(* Logix 5000 project; controller Comas_L4 vendor 1 type 14 code 193 rev 30.11; software revision 30.02; part 3 of 12 *)

ADD_ON_INSTRUCTION Message_Axe   (* revision 1.1 *)
VAR_IN_OUT
   MIO_Axis : AXIS_CIP_DRIVE; {required}
   Inf_Messages : STRING[380]; {required}
END_VAR
VAR_OUTPUT
   ER : BOOL; {access Read Only, visible}
END_VAR
VAR_IN_OUT
   Message_Defaut : STRING; {required}
   L_Msg_Index : DINT; {required}
END_VAR
VAR
   TRUE : BOOL := 1;
   FALSE : BOOL;
   L_MemoResultIndex : DINT; {access None}
   Numero_Texte : DINT; {access Read Only}
END_VAR

ROUTINE Logic   (* structured text *)
   
   	(*----------------------------------------------------------------------------------------------------
   										Build Axis ResultText String Info
   	-----------------------------------------------------------------------------------------------------*)
   		IF L_MemoResultIndex <> L_Msg_Index THEN
   			COP(Inf_Messages[L_Msg_Index],Message_Defaut,1);
   			L_MemoResultIndex					:= L_Msg_Index;
   		END_IF;
   (*================================================================================================
   										CHECK FAULT
   ==================================================================================================*)
   IF MIO_Axis.AxisFault <> 0 THEN
   
   	(*================================================================================================
   									Physical Axis Fault
   	==================================================================================================*)
   	IF MIO_Axis.AxisFault.0 THEN
   		(*================================================================================================
   										MOTOR COMMUTATION FAULT
   			==================================================================================================*)
   			IF 		MIO_Axis.MotorCommutationFault THEN
   			 		L_Msg_Index													:= 134;							// Convert INT_To_DINT
   					Numero_Texte														:= 2000+ L_Msg_Index;			// Class 2 Fault
   			(*================================================================================================
   										MOTOR OVERSEPEED FL FAULT
   			==================================================================================================*)
   			ELSIF 	MIO_Axis.MotorOverspeedFLFault THEN
   			 		L_Msg_Index													:= 135;							// Convert INT_To_DINT
   					Numero_Texte														:= 2000+ L_Msg_Index;			// Class 2 Faultt
   			(*================================================================================================
   										MOTOR OVERSEPEED UL FAULT
   			==================================================================================================*)
   			ELSIF 	MIO_Axis.MotorOverspeedULFault THEN
   			 		L_Msg_Index													:= 136;							// Convert INT_To_DINT
   					Numero_Texte														:= 2000+ L_Msg_Index;			// Class 2 Faultt
   			(*================================================================================================
   										MOTOR OVERTEMPERATURE FL FAULT
   			==================================================================================================*)
   			ELSIF 	MIO_Axis.MotorOvertemperatureFLFault THEN
   			 		L_Msg_Index													:= 137;							// Convert INT_To_DINT
   					Numero_Texte														:= 2000+ L_Msg_Index;			// Class 2 Faultt
   			(*================================================================================================
   										MOTOR OVERTEMPERATURE UL FAULT
   			==================================================================================================*)
   			ELSIF 	MIO_Axis.MotorOvertemperatureULFault THEN
   			 		L_Msg_Index													:= 138;							// Convert INT_To_DINT
   					Numero_Texte														:= 2000+ L_Msg_Index;			// Class 2 Faultt
   			(*================================================================================================
   										MOTOR THERMAL OVERLOAD FL FAULT
   			==================================================================================================*)
   			ELSIF 	MIO_Axis.MotorThermalOverloadFLFault THEN
   			 		L_Msg_Index													:= 139;							// Convert INT_To_DINT
   					Numero_Texte														:= 2000+ L_Msg_Index;			// Class 2 Faultt
   			(*================================================================================================
   										MOTOR THERMAL OVERLOAD UL FAULT
   			==================================================================================================*)
   			ELSIF 	MIO_Axis.MotorThermalOverloadULFault THEN
   			 		L_Msg_Index													:= 140;							// Convert INT_To_DINT
   					Numero_Texte														:= 2000+ L_Msg_Index;			// Class 2 Faultt
   			(*================================================================================================
   										INVERTER OVERCURRENT FAULT
   			==================================================================================================*)
   			ELSIF 	MIO_Axis.InverterOvercurrentFault THEN
   			 		L_Msg_Index													:= 141;							// Convert INT_To_DINT
   					Numero_Texte														:= 2000+ L_Msg_Index;			// Class 2 Faultt
   			(*================================================================================================
   										INVERTER OVERTEMPERATURE FL FAULT
   			==================================================================================================*)
   			ELSIF 	MIO_Axis.InverterOvertemperatureFLFault THEN
   			 		L_Msg_Index													:= 142;							// Convert INT_To_DINT
   					Numero_Texte														:= 2000+ L_Msg_Index;			// Class 2 Faultt
   			(*================================================================================================
   										INVERTER OVERTEMPERATURE UL FAULT
   			==================================================================================================*)
   			ELSIF 	MIO_Axis.InverterOvertemperatureULFault THEN
   			 		L_Msg_Index													:= 143;							// Convert INT_To_DINT
   					Numero_Texte														:= 2000+ L_Msg_Index;			// Class 2 Faultt
   			(*================================================================================================
   										INVERTER THERMALOVERLOAD FL FAULT
   			==================================================================================================*)
   			ELSIF 	MIO_Axis.InverterThermalOverloadFLFault THEN
   			 		L_Msg_Index													:= 144;							// Convert INT_To_DINT
   					Numero_Texte														:= 2000+ L_Msg_Index;			// Class 2 Faultt
   			(*================================================================================================
   										INVERTER OVERTEMPERATURE UL FAULT
   			==================================================================================================*)
   			ELSIF 	MIO_Axis.InverterOvertemperatureULFault THEN
   			 		L_Msg_Index													:= 145;							// Convert INT_To_DINT
   					Numero_Texte														:= 2000+ L_Msg_Index;			// Class 2 Faultt
   			(*================================================================================================
   										CONVERTER GROUND CURRENT FL FAULT
   			==================================================================================================*)
   			ELSIF 	MIO_Axis.ConverterGroundCurrentFLFault THEN
   			 		L_Msg_Index													:= 146;							// Convert INT_To_DINT
   					Numero_Texte														:= 2000+ L_Msg_Index;			// Class 2 Faultt
   			(*================================================================================================
   										CONVERTER GROUND CURRENT UL FAULT
   			==================================================================================================*)
   			ELSIF 	MIO_Axis.ConverterGroundCurrentULFault THEN
   			 		L_Msg_Index													:= 147;							// Convert INT_To_DINT
   					Numero_Texte														:= 2000+ L_Msg_Index;			// Class 2 Faultt
   			(*================================================================================================
   										CONVERTER OVERTEMPERATURE FL FAULT
   			==================================================================================================*)
   			ELSIF 	MIO_Axis.ConverterOvertemperatureFLFault THEN
   			 		L_Msg_Index													:= 148;							// Convert INT_To_DINT
   					Numero_Texte														:= 2000+ L_Msg_Index;			// Class 2 Faultt
   			(*================================================================================================
   										CONVERTER OVERTEMPERATURE UL FAULT
   			==================================================================================================*)
   			ELSIF 	MIO_Axis.ConverterOvertemperatureULFault THEN
   			 		L_Msg_Index													:= 149;							// Convert INT_To_DINT
   					Numero_Texte														:= 2000+ L_Msg_Index;			// Class 2 Faultt
   			(*================================================================================================
   										CONVERTER THERMAL OVERLOAD FL FAULT
   			==================================================================================================*)
   			ELSIF 	MIO_Axis.ConverterThermalOverloadFLFault THEN
   			 		L_Msg_Index													:= 150;							// Convert INT_To_DINT
   					Numero_Texte														:= 2000+ L_Msg_Index;			// Class 2 Faultt
   			(*================================================================================================
   										CONVERTER THERMAL OVERLOAD UL FAULT
   			==================================================================================================*)
   			ELSIF 	MIO_Axis.ConverterThermalOverloadULFault THEN
   			 		L_Msg_Index													:= 151;							// Convert INT_To_DINT
   					Numero_Texte														:= 2000+ L_Msg_Index;			// Class 2 Faultt
   			(*================================================================================================
   										CONVERTER AC POWER LOSS FAULT
   			==================================================================================================*)
   			ELSIF 	MIO_Axis.ConverterACPowerLossFault THEN
   			 		L_Msg_Index													:= 152;							// Convert INT_To_DINT
   					Numero_Texte														:= 2000+ L_Msg_Index;			// Class 2 Faultt
   			(*================================================================================================
   										CONVERTER AC SINGLE PHASE LOSS FAULT
   			==================================================================================================*)
   			ELSIF 	MIO_Axis.ConverterACSinglePhaseLossFault THEN
   			 		L_Msg_Index													:= 153;							// Convert INT_To_DINT
   					Numero_Texte														:= 2000+ L_Msg_Index;			// Class 2 Faultt
   			(*================================================================================================
   										CONVERTER AC PHASE SHORT FAULT
   			==================================================================================================*)
   			ELSIF 	MIO_Axis.ConverterACPhaseShortFault THEN
   			 		L_Msg_Index													:= 154;							// Convert INT_To_DINT
   					Numero_Texte														:= 2000+ L_Msg_Index;			// Class 2 Faultt
   			(*================================================================================================
   										CONVERTER PRE CHARGE FAULT
   			==================================================================================================*)
   			ELSIF 	MIO_Axis.ConverterACSinglePhaseLossFault THEN
   			 		L_Msg_Index													:= 155;							// Convert INT_To_DINT
   					Numero_Texte														:= 2000+ L_Msg_Index;			// Class 2 Faultt
   			(*================================================================================================
   										BUS REGULATOR OVERTEMPERATURE FL FAULT
   			==================================================================================================*)
   			ELSIF 	MIO_Axis.BusRegulatorOvertemperatureFLFault THEN
   			 		L_Msg_Index													:= 156;							// Convert INT_To_DINT
   					Numero_Texte														:= 2000+ L_Msg_Index;			// Class 2 Faultt
   			(*================================================================================================
   										BUS REGULATOR OVERTEMPERATURE UL FAULT
   			==================================================================================================*)
   			ELSIF 	MIO_Axis.BusRegulatorOvertemperatureULFault THEN
   			 		L_Msg_Index													:= 157;							// Convert INT_To_DINT
   					Numero_Texte														:= 2000+ L_Msg_Index;			// Class 2 Faultt
   			(*================================================================================================
   										BUS REGULATOR THERMAL OVERLOAD FL FAULT
   			==================================================================================================*)
   			ELSIF 	MIO_Axis.BusRegulatorThermalOverloadFLFault THEN
   			 		L_Msg_Index													:= 158;							// Convert INT_To_DINT
   					Numero_Texte														:= 2000+ L_Msg_Index;			// Class 2 Faultt
   			(*================================================================================================
   										BUS REGULATOR THERMAL OVERLOAD UL FAULT
   			==================================================================================================*)
   			ELSIF 	MIO_Axis.BusRegulatorThermalOverloadULFault THEN
   			 		L_Msg_Index													:= 159;							// Convert INT_To_DINT
   					Numero_Texte														:= 2000+ L_Msg_Index;			// Class 2 Faultt
   			(*================================================================================================
   										BUS UNDERVOLTAGE FL FAULT
   			==================================================================================================*)
   			ELSIF 	MIO_Axis.BusUndervoltageFLFault THEN
   			 		L_Msg_Index													:= 160;							// Convert INT_To_DINT
   					Numero_Texte														:= 2000+ L_Msg_Index;			// Class 2 Faultt
   			(*================================================================================================
   										BUS UNDERVOLTAGE UL FAULT
   			==================================================================================================*)
   			ELSIF 	MIO_Axis.BusUndervoltageULFault THEN
   			 		L_Msg_Index													:= 161;							// Convert INT_To_DINT
   					Numero_Texte														:= 2000+ L_Msg_Index;			// Class 2 Faultt
   			(*================================================================================================
   										BUS OVERVOLTAGE FL FAULT
   			==================================================================================================*)
   			ELSIF 	MIO_Axis.BusOvervoltageFLFault THEN
   			 		L_Msg_Index													:= 162;							// Convert INT_To_DINT
   					Numero_Texte														:= 2000+ L_Msg_Index;			// Class 2 Faultt
   			(*================================================================================================
   										BUS OVERVOLTAGE UL FAULT
   			==================================================================================================*)
   			ELSIF 	MIO_Axis.BusOvervoltageULFault THEN
   			 		L_Msg_Index													:= 163;							// Convert INT_To_DINT
   					Numero_Texte														:= 2000+ L_Msg_Index;			// Class 2 Faultt
   			(*================================================================================================
   										BUS POWER LOSS FAULT
   			==================================================================================================*)
   			ELSIF 	MIO_Axis.BusPowerLossFault THEN
   			 		L_Msg_Index													:= 164;							// Convert INT_To_DINT
   					Numero_Texte														:= 2000+ L_Msg_Index;			// Class 2 Faultt
   			(*================================================================================================
   										BUS POWER BLOWN FUSE FAULT
   			==================================================================================================*)
   			ELSIF 	MIO_Axis.BusPowerBlownFuseFault THEN
   			 		L_Msg_Index													:= 165;							// Convert INT_To_DINT
   					Numero_Texte														:= 2000+ L_Msg_Index;			// Class 2 Faultt
   			(*================================================================================================
   										FEEDBACK SIGNAL NOISE FL FAULT
   			==================================================================================================*)
   			ELSIF 	MIO_Axis.FeedbackSignalNoiseFLFault THEN
   			 		L_Msg_Index													:= 166;							// Convert INT_To_DINT
   					Numero_Texte														:= 2000+ L_Msg_Index;			// Class 2 Faultt
   			(*================================================================================================
   										FEEDBACK SIGNAL NOISE UL FAULT
   			==================================================================================================*)
   			ELSIF 	MIO_Axis.FeedbackSignalNoiseULFault THEN
   			 		L_Msg_Index													:= 167;							// Convert INT_To_DINT
   					Numero_Texte														:= 2000+ L_Msg_Index;			// Class 2 Faultt
   			(*================================================================================================
   										FEEDBACK SIGNAL LOSS FL FAULT
   			==================================================================================================*)
   			ELSIF 	MIO_Axis.FeedbackSignalLossFLFault THEN
   			 		L_Msg_Index													:= 168;							// Convert INT_To_DINT
   					Numero_Texte														:= 2000+ L_Msg_Index;			// Class 2 Faultt
   			(*================================================================================================
   										FEEDBACK SIGNAL LOSS UL FAULT
   			==================================================================================================*)
   			ELSIF 	MIO_Axis.FeedbackSignalLossULFault THEN
   			 		L_Msg_Index													:= 169;							// Convert INT_To_DINT
   					Numero_Texte														:= 2000+ L_Msg_Index;			// Class 2 Faultt
   			(*================================================================================================
   										FEEDBACK DATA LOSS FL FAULT
   			==================================================================================================*)
   			ELSIF 	MIO_Axis.FeedbackDataLossFLFault THEN
   			 		L_Msg_Index													:= 170;							// Convert INT_To_DINT
   					Numero_Texte														:= 2000+ L_Msg_Index;			// Class 2 Faultt
   			(*================================================================================================
   										FEEDBACK DATA LOSS UL FAULT
   			==================================================================================================*)
   			ELSIF 	MIO_Axis.FeedbackDataLossULFault THEN
   			 		L_Msg_Index													:= 171;							// Convert INT_To_DINT
   					Numero_Texte														:= 2000+ L_Msg_Index;			// Class 2 Faultt
   			(*================================================================================================
   										FEEDBACK DEVICE FAULT
   			==================================================================================================*)
   			ELSIF 	MIO_Axis.FeedbackDeviceFault THEN
   			 		L_Msg_Index													:= 172;							// Convert INT_To_DINT
   					Numero_Texte														:= 2000+ L_Msg_Index;			// Class 2 Faultt
   			(*================================================================================================
   										HARDWARE OVERTRAVEL POSITIVE FAULT
   			==================================================================================================*)
   			ELSIF 	MIO_Axis.HardwareOvertravelPositiveFault THEN
   			 		L_Msg_Index													:= 173;							// Convert INT_To_DINT
   					Numero_Texte														:= 2000+ L_Msg_Index;			// Class 2 Faultt
   			(*================================================================================================
   										HARDWARE OVERTRAVEL NEGATIVE FAULT
   			==================================================================================================*)
   			ELSIF 	MIO_Axis.HardwareOvertravelNegativeFault THEN
   			 		L_Msg_Index													:= 174;							// Convert INT_To_DINT
   					Numero_Texte														:= 2000+ L_Msg_Index;			// Class 2 Faultt
   			(*================================================================================================
   										EXCESSIVE POSITION ERROR FAULT
   			==================================================================================================*)
   			ELSIF 	MIO_Axis.ExcessivePositionErrorFault	THEN
   			 		L_Msg_Index													:= 175;							// Convert INT_To_DINT
   					Numero_Texte														:= 2000+ L_Msg_Index;			// Class 2 Faultt
   			(*================================================================================================
   										EXCESSIVE VELOCITY ERROR FAULT
   			==================================================================================================*)
   			ELSIF 	MIO_Axis.ExcessiveVelocityErrorFault	THEN
   			 		L_Msg_Index													:= 176;							// Convert INT_To_DINT
   					Numero_Texte														:= 2000+ L_Msg_Index;			// Class 2 Faultt
   			(*================================================================================================
   										OVERTORQUE LIMIT FAULT
   			==================================================================================================*)
   			ELSIF 	MIO_Axis.OvertorqueLimitFault	THEN
   			 		L_Msg_Index													:= 177;							// Convert INT_To_DINT
   					Numero_Texte														:= 2000+ L_Msg_Index;			// Class 2 Faultt
   			(*================================================================================================
   										UNDERTORQUE LIMIT FAULT
   			==================================================================================================*)
   			ELSIF 	MIO_Axis.UndertorqueLimitFault	THEN
   			 		L_Msg_Index													:= 178;							// Convert INT_To_DINT
   					Numero_Texte														:= 2000+ L_Msg_Index;			// Class 2 Faultt
   			(*================================================================================================
   										ILLEGAL CONTROL MODE FAULT
   			==================================================================================================*)
   			ELSIF 	MIO_Axis.IllegalControlModeFault	THEN
   			 		L_Msg_Index													:= 179;							// Convert INT_To_DINT
   					Numero_Texte														:= 2000+ L_Msg_Index;			// Class 2 Faultt
   			(*================================================================================================
   										ENABLE INPUT DEACTIVATED FAULT
   			==================================================================================================*)
   			ELSIF 	MIO_Axis.EnableInputDeactivatedFault	THEN
   			 		L_Msg_Index													:= 180;							// Convert INT_To_DINT
   					Numero_Texte														:= 2000+ L_Msg_Index;			// Class 2 Faultt
   			(*================================================================================================
   										CONTROLLER INITIATED FAULT
   			==================================================================================================*)
   			ELSIF 	MIO_Axis.ControllerInitiatedFault	THEN
   			 		L_Msg_Index													:= 181;							// Convert INT_To_DINT
   					Numero_Texte														:= 2000+ L_Msg_Index;			// Class 2 Faultt
   			(*================================================================================================
   										EXTERNAL INPUT FAULT
   			==================================================================================================*)
   			ELSIF 	MIO_Axis.ExternalInputFault	THEN
   			 		L_Msg_Index													:= 182;							// Convert INT_To_DINT
   					Numero_Texte														:= 2000+ L_Msg_Index;			// Class 2 Faultt
   			(*================================================================================================
   										COMMUTATION STARTUP FAULT
   			==================================================================================================*)
   			ELSIF	MIO_Axis.CommutationStartupFault THEN
   					L_Msg_Index													:= 183;							// Convert INT_To_DINT
   					Numero_Texte														:= 2000+ L_Msg_Index;			// Class 2 Faultt
   			(*================================================================================================
   										MOTOR VOLTAGE FAULT
   			==================================================================================================*)
   			ELSIF	MIO_Axis.MotorVoltageMismatchFault THEN
   					L_Msg_Index													:= 184;							// Convert INT_To_DINT
   					Numero_Texte														:= 2000+ L_Msg_Index;			// Class 2 Faultt
   			(*================================================================================================
   										FEEDBACK FILTER FAULT
   			==================================================================================================*)
   			ELSIF	MIO_Axis.FeedbackFilterNoiseFault THEN
   					L_Msg_Index													:= 185;							// Convert INT_To_DINT
   					Numero_Texte														:= 2000+ L_Msg_Index;			// Class 2 Faultt
   			(*================================================================================================
   										FEEDBACK BATTERY LOSS FAULT
   			==================================================================================================*)
   			ELSIF	MIO_Axis.FeedbackBatteryLossFault THEN
   					L_Msg_Index													:= 186;							// Convert INT_To_DINT
   					Numero_Texte														:= 2000+ L_Msg_Index;			// Class 2 Faultt
   			(*================================================================================================
   										FEEDBACK BATTERY LOW FAULT
   			==================================================================================================*)
   			ELSIF	MIO_Axis.FeedbackBatteryLowFault THEN
   					L_Msg_Index													:= 187;							// Convert INT_To_DINT
   					Numero_Texte														:= 2000+ L_Msg_Index;			// Class 2 Faultt
   			(*================================================================================================
   										FEEDBACK INCREMENTAL COUNT FAULT
   			==================================================================================================*)
   			ELSIF	MIO_Axis.FeedbackIncrementalCountErrorFault THEN
   					L_Msg_Index													:= 188;							// Convert INT_To_DINT
   					Numero_Texte														:= 2000+ L_Msg_Index;			// Class 2 Faultt
   			(*================================================================================================
   										CONTROL MODULE OVT FACTORY FAULT
   			==================================================================================================*)
   			ELSIF	MIO_Axis.ControlModuleOvertemperatureFLFault THEN
   					L_Msg_Index													:= 189;							// Convert INT_To_DINT
   					Numero_Texte														:= 2000+ L_Msg_Index;			// Class 2 Faultt
   			(*================================================================================================
   										CONTROL MODULE OVT USER FAULT
   			==================================================================================================*)
   			ELSIF	MIO_Axis.ControlModuleOvertemperatureULFault THEN
   					L_Msg_Index													:= 190;							// Convert INT_To_DINT
   					Numero_Texte														:= 2000+ L_Msg_Index;			// Class 2 Faultt
   			(*================================================================================================
   										CONVERTER PRECHARGE OVERLOAD FACTORY FAULT
   			==================================================================================================*)
   			ELSIF	MIO_Axis.ConverterPreChargeOverloadFLFault THEN
   					L_Msg_Index													:= 191;							// Convert INT_To_DINT
   					Numero_Texte														:= 2000+ L_Msg_Index;			// Class 2 Faultt
   			(*================================================================================================
   										CONVERTER PRECHARGE OVERLOAD USER FAULT
   			==================================================================================================*)
   			ELSIF	MIO_Axis.ConverterPreChargeOverloadULFault THEN
   					L_Msg_Index													:= 192;							// Convert INT_To_DINT
   					Numero_Texte														:= 2000+ L_Msg_Index;			// Class 2 Faultt
   			(*================================================================================================
   										CURRENT FEEDBACK FAULT
   			==================================================================================================*)
   			ELSIF	MIO_Axis.ExcessiveCurrentFeedbackOffsetFault THEN
   					L_Msg_Index													:= 193;							// Convert INT_To_DINT
   					Numero_Texte														:= 2000+ L_Msg_Index;			// Class 2 Faultt
   			(*================================================================================================
   										REGENERATIVE POWER SUPPLY FAULT
   			==================================================================================================*)
   			ELSIF	MIO_Axis.RegenerativePowerSupplyFault THEN
   					L_Msg_Index													:= 194;							// Convert INT_To_DINT
   					Numero_Texte														:= 2000+ L_Msg_Index;			// Class 2 Faultt
   			(*================================================================================================
   										PWR FREQUENCY REDUCED FAULT
   			==================================================================================================*)
   			ELSIF	MIO_Axis.PWMFrequencyReducedFault THEN
   					L_Msg_Index													:= 195;							// Convert INT_To_DINT
   					Numero_Texte														:= 2000+ L_Msg_Index;			// Class 2 Faultt
   			(*================================================================================================
   										CURRENT LIMIT REDUCED FAULT
   			==================================================================================================*)
   			ELSIF	MIO_Axis.CurrentLimitReducedFault THEN
   					L_Msg_Index													:= 196;							// Convert INT_To_DINT
   					Numero_Texte														:= 2000+ L_Msg_Index;			// Class 2 Faultt
   			(*================================================================================================
   										TORQUE PROVE FAULT
   			==================================================================================================*)
   			ELSIF	MIO_Axis.TorqueProveFault THEN
   					L_Msg_Index													:= 197;							// Convert INT_To_DINT
   					Numero_Texte														:= 2000+ L_Msg_Index;			// Class 2 Faultt
   			(*================================================================================================
   										DECEL OVERRIDE FAULT
   			==================================================================================================*)
   			ELSIF	MIO_Axis.DecelOverrideFault THEN
   					L_Msg_Index													:= 198;							// Convert INT_To_DINT
   					Numero_Texte														:= 2000+ L_Msg_Index;			// Class 2 Faultt
   			(*================================================================================================
   										PREVENTIVE MAINTENANCE FAULT
   			==================================================================================================*)
   			ELSIF	MIO_Axis.PreventativeMaintenanceFault THEN
   					L_Msg_Index													:= 199;							// Convert INT_To_DINT
   					Numero_Texte														:= 2000+ L_Msg_Index;			// Class 2 Faultt
   			(*================================================================================================
   										MOTOR TEST FAULT
   			==================================================================================================*)
   			ELSIF	MIO_Axis.MotorTestFault THEN
   					L_Msg_Index													:= 240;							// Convert INT_To_DINT
   					Numero_Texte														:= 2000+ L_Msg_Index;			// Class 2 Faultt
   			(*================================================================================================
   										HARDWARE CONFIGURATION FAULT
   			==================================================================================================*)
   			ELSIF	MIO_Axis.HardwareConfigurationFault THEN
   					L_Msg_Index													:= 241;							// Convert INT_To_DINT
   					Numero_Texte														:= 2000+ L_Msg_Index;			// Class 2 Faultt
   			(*================================================================================================
   										FIRMWARE CONFIGURATION FAULT
   			==================================================================================================*)
   			ELSIF	MIO_Axis.FirmwareChangeFault THEN
   					L_Msg_Index													:= 242;							// Convert INT_To_DINT
   					Numero_Texte														:= 2000+ L_Msg_Index;			// Class 2 Faultt
   			(*================================================================================================
   										DC COMMON BUS FAULT
   			==================================================================================================*)
   			ELSIF	MIO_Axis.DCCommonBusFault THEN
   					L_Msg_Index													:= 243;							// Convert INT_To_DINT
   					Numero_Texte														:= 2000+ L_Msg_Index;			// Class 2 Faultt
   			(*================================================================================================
   										RUNTIME ERROR FAULT
   			==================================================================================================*)
   			ELSIF	MIO_Axis.RuntimeErrorFault THEN
   					L_Msg_Index													:= 244;							// Convert INT_To_DINT
   					Numero_Texte														:= 2000+ L_Msg_Index;			// Class 2 Faultt
   			(*================================================================================================
   										BACKPLANE COMMUNICATION ERROR FAULT
   			==================================================================================================*)
   			ELSIF	MIO_Axis.BackplaneCommunicationErrorFault THEN
   					L_Msg_Index													:= 245;							// Convert INT_To_DINT
   					Numero_Texte														:= 2000+ L_Msg_Index;			// Class 2 Faultt
   			(*================================================================================================
   										SAFETY MODULE COMMUNICATION ERROR FAULT
   			==================================================================================================*)
   			ELSIF	MIO_Axis.SafetyModuleCommunicationErrorFault THEN
   					L_Msg_Index													:= 246;							// Convert INT_To_DINT
   					Numero_Texte														:= 2000+ L_Msg_Index;			// Class 2 Faultt
   			(*================================================================================================
   										PRODUCT SPECIFIC FAULT
   			==================================================================================================*)
   			ELSIF	MIO_Axis.ProductSpecificFault THEN
   					L_Msg_Index													:= 247;							// Convert INT_To_DINT
   					Numero_Texte														:= 2000+ L_Msg_Index;			// Class 2 Faultt
   			END_IF;
   
   	(*================================================================================================
   									Module Fault
   	==================================================================================================*)
   	ELSIF MIO_Axis.AxisFault.1 THEN
   			(*================================================================================================
   										CONTROL SYNC FAULT
   			==================================================================================================*)
   			IF 		MIO_Axis.ControlSyncFault THEN
   					L_Msg_Index													:= 250;
   					Numero_Texte														:= 1000 + L_Msg_Index;		// Class 1 Fault
   			(*================================================================================================
   										MODULE SYNC FAULT
   			==================================================================================================*)
   			ELSIF 	MIO_Axis.ModuleSyncFault THEN
   					L_Msg_Index													:= 251;
   					Numero_Texte														:= 1000 + L_Msg_Index;		// Class 1 Fault
   			(*================================================================================================
   										TIMER EVENT FAULT
   			==================================================================================================*)
   			ELSIF 	MIO_Axis.TimerEventFault THEN
   					L_Msg_Index													:= 252;
   					Numero_Texte														:= 1000 + L_Msg_Index;		// Class 1 Fault
   			(*================================================================================================
   										MODULE HARDWARE FAULT
   			==================================================================================================*)
   			ELSIF 	MIO_Axis.ModuleHardwareFault THEN
   					L_Msg_Index													:= 253;
   					Numero_Texte														:= 1000 + L_Msg_Index;		// Class 1 Fault
   			(*================================================================================================
   										MODULE CONNECTION FAULT
   			==================================================================================================*)
   			ELSIF 	MIO_Axis.ModuleConnFault THEN
   					L_Msg_Index													:= 254;
   					Numero_Texte														:= 1000 + L_Msg_Index;		// Class 1 Fault
   			(*================================================================================================
   										CONNEXION FORMAT FAULT
   			==================================================================================================*)
   			ELSIF	MIO_Axis.ConnFormatFault THEN
   					L_Msg_Index													:= 255;
   					Numero_Texte														:= 1000 + L_Msg_Index;		// Class 1 Fault
   			(*================================================================================================
   										LOCAL MODE FAULT
   			==================================================================================================*)
   			ELSIF 	MIO_Axis.LocalModeFault THEN
   					L_Msg_Index													:= 256;
   					Numero_Texte														:= 1000 + L_Msg_Index;		// Class 1 Fault
   			(*================================================================================================
   										CPU WATCHDOG FAULT
   			==================================================================================================*)
   			ELSIF 	MIO_Axis.CPUWatchdogFault THEN
   					L_Msg_Index													:= 257;
   					Numero_Texte														:= 1000 + L_Msg_Index;		// Class 1 Fault
   			(*================================================================================================
   										CLOCK JITTER FAULT
   			==================================================================================================*)
   			ELSIF 	MIO_Axis.ClockJitterFault THEN
   					L_Msg_Index													:= 258;
   					Numero_Texte														:= 1000 + L_Msg_Index;		// Class 1 Fault
   			(*================================================================================================
   										CYCLIC READ FAULT
   			==================================================================================================*)
   			ELSIF 	MIO_Axis.CyclicReadFault THEN
   					L_Msg_Index													:= 259;
   					Numero_Texte														:= 1000 + L_Msg_Index;		// Class 1 Fault
   			(*================================================================================================
   										CYCLIC WRITE FAULT
   			==================================================================================================*)
   			ELSIF 	MIO_Axis.CyclicWriteFault THEN
   					L_Msg_Index													:= 260;
   					Numero_Texte														:= 1000 + L_Msg_Index;		// Class 1 Fault
   			(*================================================================================================
   										CLOCK SKEW FAULT
   			==================================================================================================*)
   			ELSIF 	MIO_Axis.ClockSkewFault THEN
   					L_Msg_Index													:= 261;
   					Numero_Texte														:= 1000 + L_Msg_Index;		// Class 1 Fault
   			(*================================================================================================
   										CONTROL CONNEXION FAULT
   			==================================================================================================*)
   			ELSIF 	MIO_Axis.ControlConnFault THEN
   					L_Msg_Index													:= 262;
   					Numero_Texte														:= 1000 + L_Msg_Index;		// Class 1 Fault
   			(*================================================================================================
   										CONTROL CLOCK SYNC FAULT
   										Correction CLG
   										MIO_Axis.ControlClockSyncFault -> MIO_Axis.ClockSyncFault
   			==================================================================================================*)
   			ELSIF 	MIO_Axis.ClockSyncFault THEN
   					L_Msg_Index													:= 263;
   					Numero_Texte														:= 1000 + L_Msg_Index;		// Class 1 Fault
   			(*================================================================================================
   										MODULE CLOCK SYNC FAULT
   										Correction CLG
   										Deleted
   			==================================================================================================*)
   			(*ELSIF 	MIO_Axis.ModuleClockSyncFault THEN
   					L_ResultIndex													:= 264;
   					Sts_Result														:= 1000 + L_ResultIndex;		// Class 1 Fault
   			(*================================================================================================
   										LOGIC WATCHDOG FAULT
   			==================================================================================================*)
   			ELSIF 	MIO_Axis.LogicWatchdogFault THEN
   					L_Msg_Index													:= 265;
   					Numero_Texte														:= 1000 + L_Msg_Index;		// Class 1 Fault
   			(*================================================================================================
   										DUPLICATE ADRESS FAULT
   			==================================================================================================*)
   			ELSIF 	MIO_Axis.DuplicateAddressFault THEN
   					L_Msg_Index													:= 266;
   					Numero_Texte														:= 1000 + L_Msg_Index;		// Class 1 Fault
   			END_IF;
   
   	(*================================================================================================
   									Configuration Fault
   	==================================================================================================*)
   	ELSIF MIO_Axis.AxisFault.2 THEN
   
   		 	CASE MIO_Axis.AttributeErrorCode OF
   
   			(*================================================================================================
   										Connection failure
   			==================================================================================================*)
   			1 :		L_Msg_Index													:= 270;
   					Numero_Texte														:= 1000 + L_Msg_Index;		// Class 1 Fault
   			(*================================================================================================
   										Ressource unavalaible
   			==================================================================================================*)
   			2 :		L_Msg_Index													:= 271;
   					Numero_Texte														:= 1000 + L_Msg_Index;		// Class 1 Fault
   			(*================================================================================================
   										Invalid value in object specific datab parameter of a service request.
   			==================================================================================================*)
   			3 :		L_Msg_Index													:= 272;
   					Numero_Texte														:= 1000 + L_Msg_Index;		// Class 1 Fault
   			(*================================================================================================
   										IOI segment error.
   			==================================================================================================*)
   			4 :		L_Msg_Index													:= 273;
   					Numero_Texte														:= 1000 + L_Msg_Index;		// Class 1 Fault
   			(*================================================================================================
   										IOI destination unknown.
   			==================================================================================================*)
   			5 :		L_Msg_Index													:= 274;
   					Numero_Texte														:= 1000 + L_Msg_Index;		// Class 1 Fault
   			(*================================================================================================
   										Partial transfer.
   			==================================================================================================*)
   			6 :		L_Msg_Index													:= 275;
   					Numero_Texte														:= 1000 + L_Msg_Index;		// Class 1 Fault
   			(*================================================================================================
   										Connection lost.
   			==================================================================================================*)
   			7 :		L_Msg_Index													:= 276;
   					Numero_Texte														:= 1000 + L_Msg_Index;		// Class 1 Fault
   			(*================================================================================================
   										Unimplemented service.
   			==================================================================================================*)
   			8 :		L_Msg_Index													:= 277;
   					Numero_Texte														:= 1000 + L_Msg_Index;		// Class 1 Fault
   			(*================================================================================================
   										Invalid attribute value.
   			==================================================================================================*)
   			9 :		L_Msg_Index													:= 278;
   					Numero_Texte														:= 1000 + L_Msg_Index;		// Class 1 Fault
   			(*================================================================================================
   										Attribute list error.
   			==================================================================================================*)
   			10 :	L_Msg_Index													:= 279;
   					Numero_Texte														:= 1000 + L_Msg_Index;		// Class 1 Fault
   			(*================================================================================================
   										Already in requested mode/state.
   			==================================================================================================*)
   			11 :	L_Msg_Index													:= 280;
   					Numero_Texte														:= 1000 + L_Msg_Index;		// Class 1 Fault
   			(*================================================================================================
   										Object can not perform service in its current mode/state.
   			==================================================================================================*)
   			12 :	L_Msg_Index													:= 281;
   					Numero_Texte														:= 1000 + L_Msg_Index;		// Class 1 Fault
   			(*================================================================================================
   										Object already exists.
   			==================================================================================================*)
   			13 :	L_Msg_Index													:= 282;
   					Numero_Texte														:= 1000 + L_Msg_Index;		// Class 1 Fault
   			(*================================================================================================
   										Attribute value not settable.
   			==================================================================================================*)
   			14 :	L_Msg_Index													:= 283;
   					Numero_Texte														:= 1000 + L_Msg_Index;		// Class 1 Fault
   			(*================================================================================================
   										Access permission does not allow service.
   			==================================================================================================*)
   			15 :	L_Msg_Index													:= 284;
   					Numero_Texte														:= 1000 + L_Msg_Index;		// Class 1 Fault
   			(*================================================================================================
   										Device’s mode/state does not allow object to perform service.
   			==================================================================================================*)
   			16 :	L_Msg_Index													:= 285;
   					Numero_Texte														:= 1000 + L_Msg_Index;		// Class 1 Fault
   			(*================================================================================================
   										Reply data too large.
   			==================================================================================================*)
   			17 :	L_Msg_Index													:= 286;
   					Numero_Texte														:= 1000 + L_Msg_Index;		// Class 1 Fault
   			(*================================================================================================
   										Fragmentation of a primitive value.
   			==================================================================================================*)
   			18 :	L_Msg_Index													:= 287;
   					Numero_Texte														:= 1000 + L_Msg_Index;		// Class 1 Fault
   			(*================================================================================================
   										Not enough data.
   			==================================================================================================*)
   			19 :	L_Msg_Index													:= 288;
   					Numero_Texte														:= 1000 + L_Msg_Index;		// Class 1 Fault
   			(*================================================================================================
   										Undefined attribute.
   			==================================================================================================*)
   			20 :	L_Msg_Index													:= 289;
   					Numero_Texte														:= 1000 + L_Msg_Index;		// Class 1 Fault
   			(*================================================================================================
   										Too much data.
   			==================================================================================================*)
   			21 :	L_Msg_Index													:= 290;
   					Numero_Texte														:= 1000 + L_Msg_Index;		// Class 1 Fault
   			(*================================================================================================
   										Object does not exist.
   			==================================================================================================*)
   			22 :	L_Msg_Index													:= 291;
   					Numero_Texte														:= 1000 + L_Msg_Index;		// Class 1 Fault
   			(*================================================================================================
   										Service fragmentation sequence not
   										currently in progress.
   			==================================================================================================*)
   			23 :	L_Msg_Index													:= 292;
   					Numero_Texte														:= 1000 + L_Msg_Index;		// Class 1 Fault
   			(*================================================================================================
   										No stored attribute data.
   			==================================================================================================*)
   			24 :	L_Msg_Index													:= 293;
   					Numero_Texte														:= 1000 + L_Msg_Index;		// Class 1 Fault
   			(*================================================================================================
   										Store operation failure.
   			==================================================================================================*)
   			25 :	L_Msg_Index													:= 294;
   					Numero_Texte														:= 1000 + L_Msg_Index;		// Class 1 Fault
   			(*================================================================================================
   										Bridging failure, request packet too large for network.
   			==================================================================================================*)
   			26 :	L_Msg_Index													:= 295;
   					Numero_Texte														:= 1000 + L_Msg_Index;		// Class 1 Fault
   			(*================================================================================================
   										Bridging failure, response packet too large for network.
   			==================================================================================================*)
   			27 :	L_Msg_Index													:= 296;
   					Numero_Texte														:= 1000 + L_Msg_Index;		// Class 1 Fault
   			(*================================================================================================
   										Missing attribute list entry data.
   			==================================================================================================*)
   			28 :	L_Msg_Index													:= 297;
   					Numero_Texte														:= 1000 + L_Msg_Index;		// Class 1 Fault
   			(*================================================================================================
   										Invalid attribute value list.
   			==================================================================================================*)
   			29 :	L_Msg_Index													:= 298;
   					Numero_Texte														:= 1000 + L_Msg_Index;		// Class 1 Fault
   			(*================================================================================================
   										Embedded service error.
   			==================================================================================================*)
   			30 :	L_Msg_Index													:= 299;
   					Numero_Texte														:= 1000 + L_Msg_Index;		// Class 1 Fault
   			(*================================================================================================
   										Connection Related Failure.
   			==================================================================================================*)
   			31 :	L_Msg_Index													:= 300;
   					Numero_Texte														:= 1000 + L_Msg_Index;		// Class 1 Fault
   			(*================================================================================================
   										Invalid Parameter.
   			==================================================================================================*)
   			32 :	L_Msg_Index													:= 301;
   					Numero_Texte														:= 1000 + L_Msg_Index;		// Class 1 Fault
   			(*================================================================================================
   										Write–once value or medium already written.
   			==================================================================================================*)
   			33 :	L_Msg_Index													:= 302;
   					Numero_Texte														:= 1000 + L_Msg_Index;		// Class 1 Fault
   			(*================================================================================================
   										Invalid Reply Received.
   			==================================================================================================*)
   			34 :	L_Msg_Index													:= 303;
   					Numero_Texte														:= 1000 + L_Msg_Index;		// Class 1 Faul
   			(*================================================================================================
   										CST not coordinated.
   			==================================================================================================*)
   			35 :	L_Msg_Index													:= 304;
   					Numero_Texte														:= 1000 + L_Msg_Index;		// Class 1 Fault
   			(*================================================================================================
   										Connection Scheduling Error.
   			==================================================================================================*)
   			36 :	L_Msg_Index													:= 305;
   					Numero_Texte														:= 1000 + L_Msg_Index;		// Class 1 Fault
   			(*================================================================================================
   										Key Failure in IOI.
   			==================================================================================================*)
   			37 :	L_Msg_Index													:= 306;
   					Numero_Texte														:= 1000 + L_Msg_Index;		// Class 1 Fault
   			(*================================================================================================
   										IOI Size Invalid.
   			==================================================================================================*)
   			38 :	L_Msg_Index													:= 307;
   					Numero_Texte														:= 1000 + L_Msg_Index;		// Class 1 Fault
   			(*================================================================================================
   										Unexpected attribute in list.
   			==================================================================================================*)
   			39 :	L_Msg_Index													:= 308;
   					Numero_Texte														:= 1000 + L_Msg_Index;		// Class 1 Fault
   			(*================================================================================================
   										DNet Invalid Member ID.
   			==================================================================================================*)
   			40 :	L_Msg_Index													:= 309;
   					Numero_Texte														:= 1000 + L_Msg_Index;		// Class 1 Fault
   			(*================================================================================================
   										DNet Member not settable.
   			==================================================================================================*)
   			41 :	L_Msg_Index													:= 310;
   					Numero_Texte														:= 1000 + L_Msg_Index;		// Class 1 Fault
   			END_CASE;
   
   	(*================================================================================================
   									Group Fault
   	==================================================================================================*)
   	ELSIF MIO_Axis.AxisFault.3 THEN
   
   					L_Msg_Index													:= 311;
   					Numero_Texte														:= 1000 + L_Msg_Index;		// Class 1 Fault
   
   	(*================================================================================================
   									Motion Fault
   	==================================================================================================*)
   	ELSIF MIO_Axis.AxisFault.4 THEN
   
   			(*================================================================================================
   										POSITIVE SOFT TRAVEL LIMIT FAULT
   			==================================================================================================*)
   			IF 		MIO_Axis.SoftTravelLimitPositiveFault THEN
   			 		L_Msg_Index													:= 100;							// Convert INT_To_DINT
   					Numero_Texte														:= 2000+ L_Msg_Index;			// Class 2 Faultt
   			(*================================================================================================
   										NEGATIVE SOFT TRAVEL LIMIT FAULT
   			==================================================================================================*)
   			ELSIF 	MIO_Axis.SoftTravelLimitNegativeFault THEN
   			 		L_Msg_Index													:= 101;							// Convert INT_To_DINT
   					Numero_Texte														:= 2000+ L_Msg_Index;			// Class 2 Faultt
   			END_IF;
   
   	(*================================================================================================
   									Guard Fault
   	==================================================================================================*)
   	ELSIF MIO_Axis.AxisFault.5 THEN
   
   			(*================================================================================================
   										GUARD INTERNAL FAULT
   			==================================================================================================*)
   			IF 		MIO_Axis.GuardInternalFault THEN
   			 		L_Msg_Index													:= 312;							// Convert INT_To_DINT
   					Numero_Texte														:= 2000+ L_Msg_Index;			// Class 2 Faultt
   			(*================================================================================================
   										GUARD CONFIGURATION FAULT
   			==================================================================================================*)
   			ELSIF 	MIO_Axis.GuardConfigurationFault THEN
   			 		L_Msg_Index													:= 313;							// Convert INT_To_DINT
   					Numero_Texte														:= 2000+ L_Msg_Index;			// Class 2 Faultt
   			(*================================================================================================
   										GUARD GATE DRIVE FAULT
   			==================================================================================================*)
   			ELSIF 	MIO_Axis.GuardGateDriveFault THEN
   			 		L_Msg_Index													:= 314;							// Convert INT_To_DINT
   					Numero_Texte														:= 2000+ L_Msg_Index;			// Class 2 Faultt
   			(*================================================================================================
   										GUARD RESET FAULT
   			==================================================================================================*)
   			ELSIF 	MIO_Axis.GuardResetFault THEN
   			 		L_Msg_Index													:= 315;							// Convert INT_To_DINT
   					Numero_Texte														:= 2000+ L_Msg_Index;			// Class 2 Faultt
   			(*================================================================================================
   										GUARD FEEDBACK 1 FAULT
   			==================================================================================================*)
   			ELSIF 	MIO_Axis.GuardFeedback1Fault THEN
   			 		L_Msg_Index													:= 316;							// Convert INT_To_DINT
   					Numero_Texte														:= 2000+ L_Msg_Index;			// Class 2 Faultt
   			(*================================================================================================
   										GUARD FEEDBACK 2 FAULT
   			==================================================================================================*)
   			ELSIF 	MIO_Axis.GuardFeedback2Fault THEN
   			 		L_Msg_Index													:= 317;							// Convert INT_To_DINT
   					Numero_Texte														:= 2000+ L_Msg_Index;			// Class 2 Faultt
   			(*================================================================================================
   										GUARD FEEDBACK SPEED COMP FAULT
   			==================================================================================================*)
   			ELSIF 	MIO_Axis.GuardFeedbackSpeedCompareFault THEN
   			 		L_Msg_Index													:= 318;							// Convert INT_To_DINT
   					Numero_Texte														:= 2000+ L_Msg_Index;			// Class 2 Faultt
   			(*================================================================================================
   										GUARD FEEDBACK POSITION COMP FAULT
   			==================================================================================================*)
   			ELSIF 	MIO_Axis.GuardFeedbackPositionCompareFault THEN
   			 		L_Msg_Index													:= 319;							// Convert INT_To_DINT
   					Numero_Texte														:= 2000+ L_Msg_Index;			// Class 2 Faultt
   			(*================================================================================================
   										GUARD STOP INPUT FAULT
   			==================================================================================================*)
   			ELSIF 	MIO_Axis.GuardStopInputFault THEN
   			 		L_Msg_Index													:= 320;							// Convert INT_To_DINT
   					Numero_Texte														:= 2000+ L_Msg_Index;			// Class 2 Faultt
   			(*================================================================================================
   										GUARD STOP OUTPUT FAULT
   			==================================================================================================*)
   			ELSIF 	MIO_Axis.GuardStopOutputFault THEN
   			 		L_Msg_Index													:= 321;							// Convert INT_To_DINT
   					Numero_Texte														:= 2000+ L_Msg_Index;			// Class 2 Faultt
   			(*================================================================================================
   										GUARD STOP DECEL FAULT
   			==================================================================================================*)
   			ELSIF 	MIO_Axis.GuardStopDecelFault THEN
   			 		L_Msg_Index													:= 322;							// Convert INT_To_DINT
   					Numero_Texte														:= 2000+ L_Msg_Index;			// Class 2 Faultt
   			(*================================================================================================
   										GUARD STOP STANDSTILL FAULT
   			==================================================================================================*)
   			ELSIF 	MIO_Axis.GuardStopStandstillFault THEN
   			 		L_Msg_Index													:= 323;							// Convert INT_To_DINT
   					Numero_Texte														:= 2000+ L_Msg_Index;			// Class 2 Faultt
   			(*================================================================================================
   										GUARD STOP MOTION FAULT
   			==================================================================================================*)
   			ELSIF 	MIO_Axis.GuardStopMotionFault THEN
   			 		L_Msg_Index													:= 324;							// Convert INT_To_DINT
   					Numero_Texte														:= 2000+ L_Msg_Index;			// Class 2 Faultt
   			(*================================================================================================
   										GUARD LIMITED SPEED INPUT FAULT
   			==================================================================================================*)
   			ELSIF 	MIO_Axis.GuardLimitedSpeedInputFault THEN
   			 		L_Msg_Index													:= 325;							// Convert INT_To_DINT
   					Numero_Texte														:= 2000+ L_Msg_Index;			// Class 2 Faultt
   			(*================================================================================================
   										GUARD LIMITED SPEED OUTPUT FAULT
   			==================================================================================================*)
   			ELSIF 	MIO_Axis.GuardLimitedSpeedOutputFault THEN
   			 		L_Msg_Index													:= 326;							// Convert INT_To_DINT
   					Numero_Texte														:= 2000+ L_Msg_Index;			// Class 2 Faultt
   			(*================================================================================================
   										GUARD LIMITED SPEED MONITOR FAULT
   			==================================================================================================*)
   			ELSIF 	MIO_Axis.GuardLimitedSpeedMonitorFault THEN
   			 		L_Msg_Index													:= 327;							// Convert INT_To_DINT
   					Numero_Texte														:= 2000+ L_Msg_Index;			// Class 2 Faultt
   			(*================================================================================================
   										GUARD MAX SPEED FAULT
   			==================================================================================================*)
   			ELSIF 	MIO_Axis.GuardMaxSpeedMonitorFault THEN
   			 		L_Msg_Index													:= 328;							// Convert INT_To_DINT
   					Numero_Texte														:= 2000+ L_Msg_Index;			// Class 2 Faultt
   			(*================================================================================================
   										GUARD MAX ACCEL FAULT
   			==================================================================================================*)
   			ELSIF 	MIO_Axis.GuardMaxAccelMonitorFault THEN
   			 		L_Msg_Index													:= 329;							// Convert INT_To_DINT
   					Numero_Texte														:= 2000+ L_Msg_Index;			// Class 2 Faultt
   			(*================================================================================================
   										GUARD DIRECTION MONITOR FAULT
   			==================================================================================================*)
   			ELSIF 	MIO_Axis.GuardDirectionMonitorFault THEN
   			 		L_Msg_Index													:= 330;							// Convert INT_To_DINT
   					Numero_Texte														:= 2000+ L_Msg_Index;			// Class 2 Faultt
   			(*================================================================================================
   										GUARD DOOR MONITOR INPUT FAULT
   			==================================================================================================*)
   			ELSIF 	MIO_Axis.GuardDoorMonitorInputFault THEN
   			 		L_Msg_Index													:= 331;							// Convert INT_To_DINT
   					Numero_Texte														:= 2000+ L_Msg_Index;			// Class 2 Faultt
   			(*================================================================================================
   										GUARD DOOR MONITOR FAULT
   			==================================================================================================*)
   			ELSIF 	MIO_Axis.GuardDoorMonitorFault THEN
   			 		L_Msg_Index													:= 332;							// Convert INT_To_DINT
   					Numero_Texte														:= 2000+ L_Msg_Index;			// Class 2 Faultt
   			(*================================================================================================
   										GUARD DOOR CONTROL OUTPUT FAULT
   			==================================================================================================*)
   			ELSIF 	MIO_Axis.GuardDoorControlOutputFault THEN
   			 		L_Msg_Index													:= 333;							// Convert INT_To_DINT
   					Numero_Texte														:= 2000+ L_Msg_Index;			// Class 2 Faultt
   			(*================================================================================================
   										GUARD LOCK MONITOR INPUT FAULT
   			==================================================================================================*)
   			ELSIF 	MIO_Axis.GuardLockMonitorInputFault THEN
   			 		L_Msg_Index													:= 334;							// Convert INT_To_DINT
   					Numero_Texte														:= 2000+ L_Msg_Index;			// Class 2 Faultt
   			(*================================================================================================
   										GUARD LOCK MONITOR FAULT
   			==================================================================================================*)
   			ELSIF 	MIO_Axis.GuardLockMonitorFault THEN
   			 		L_Msg_Index													:= 335;							// Convert INT_To_DINT
   					Numero_Texte														:= 2000+ L_Msg_Index;			// Class 2 Faultt
   			(*================================================================================================
   										GUARD SWITCH MONITOR INPUT FAULT
   			==================================================================================================*)
   			ELSIF 	MIO_Axis.GuardEnablingSwitchMonitorInputFault THEN
   			 		L_Msg_Index													:= 336;							// Convert INT_To_DINT
   					Numero_Texte														:= 2000+ L_Msg_Index;			// Class 2 Faultt
   			(*================================================================================================
   										GUARD SWITCH MONITOR FAULT
   			==================================================================================================*)
   			ELSIF 	MIO_Axis.GuardEnablingSwitchMonitorFault THEN
   			 		L_Msg_Index													:= 337;							// Convert INT_To_DINT
   					Numero_Texte														:= 2000+ L_Msg_Index;			// Class 2 Faultt
   			(*================================================================================================
   										GUARD FEEDBACK 1 VOLTAGE MONITOR FAULT
   			==================================================================================================*)
   			ELSIF 	MIO_Axis.GuardFeedback1VoltageMonitorFault THEN
   			 		L_Msg_Index													:= 338;							// Convert INT_To_DINT
   					Numero_Texte														:= 2000+ L_Msg_Index;			// Class 2 Faultt
   			(*================================================================================================
   										GUARD FEEDBACK 2 VOLTAGE MONITOR FAULT
   			==================================================================================================*)
   			ELSIF 	MIO_Axis.GuardFeedback2VoltageMonitorFault THEN
   			 		L_Msg_Index													:= 339;							// Convert INT_To_DINT
   					Numero_Texte														:= 2000+ L_Msg_Index;			// Class 2 Faultt
   			END_IF;
   
   	(*================================================================================================
   									Initialisation Fault
   	==================================================================================================*)
   	ELSIF MIO_Axis.AxisFault.5 THEN
   
   			(*================================================================================================
   										Boot Block Checksum Fault
   			==================================================================================================*)
   			IF 		MIO_Axis.BootBlockChecksumFault THEN
   			 		L_Msg_Index													:= 340;							// Convert INT_To_DINT
   					Numero_Texte														:= 2000+ L_Msg_Index;			// Class 2 Faultt
   			(*================================================================================================
   										Main Block Checksum Fault
   			==================================================================================================*)
   			ELSIF 	MIO_Axis.MainBlockChecksumFault THEN
   			 		L_Msg_Index													:= 341;							// Convert INT_To_DINT
   					Numero_Texte														:= 2000+ L_Msg_Index;			// Class 2 Faultt
   			(*================================================================================================
   										Nonvolatile Memory Checksum Fault
   			==================================================================================================*)
   			ELSIF 	MIO_Axis.NonvolatileMemoryChecksumFault THEN
   			 		L_Msg_Index													:= 342;							// Convert INT_To_DINT
   					Numero_Texte														:= 2000+ L_Msg_Index;			// Class 2 Faultt
   			(*================================================================================================
   										Commutation Not Configured
   			==================================================================================================*)
   			ELSIF 	MIO_Axis.CommutationNotConfigured THEN
   			 		L_Msg_Index													:= 343;							// Convert INT_To_DINT
   					Numero_Texte														:= 2000+ L_Msg_Index;			// Class 2 Faultt
   			(*================================================================================================
   										Feedback Data Corruption
   			==================================================================================================*)
   			ELSIF 	MIO_Axis.FeedbackDataCorruptionFault THEN
   			 		L_Msg_Index													:= 344;							// Convert INT_To_DINT
   					Numero_Texte														:= 2000+ L_Msg_Index;			// Class 2 Faultt
   			(*================================================================================================
   										Feedback Data Range
   			==================================================================================================*)
   			ELSIF 	MIO_Axis.FeedbackDataRangeFault THEN
   			 		L_Msg_Index													:= 345;							// Convert INT_To_DINT
   					Numero_Texte														:= 2000+ L_Msg_Index;			// Class 2 Faultt
   			(*================================================================================================
   										Feedback Communication Startup
   			==================================================================================================*)
   			ELSIF 	MIO_Axis.FeedbackCommunicationStartupFault THEN
   			 		L_Msg_Index													:= 346;							// Convert INT_To_DINT
   					Numero_Texte														:= 2000+ L_Msg_Index;			// Class 2 Faultt
   			(*================================================================================================
   										Feedback Absolute Overspeed
   			==================================================================================================*)
   			ELSIF 	MIO_Axis.FeedbackAbsoluteOverspeedFault THEN
   			 		L_Msg_Index													:= 347;							// Convert INT_To_DINT
   					Numero_Texte														:= 2000+ L_Msg_Index;			// Class 2 Faultt
   			(*================================================================================================
   										Feedback Absolute Power Off Travel
   			==================================================================================================*)
   			ELSIF 	MIO_Axis.FeedbackAbsolutePowerOffTravelFault THEN
   			 		L_Msg_Index													:= 348;							// Convert INT_To_DINT
   					Numero_Texte														:= 2000+ L_Msg_Index;			// Class 2 Faultt
   			(*================================================================================================
   										Feedback Absolute Startup Speed
   			==================================================================================================*)
   			ELSIF 	MIO_Axis.FeedbackAbsoluteStartupSpeedFault THEN
   			 		L_Msg_Index													:= 349;							// Convert INT_To_DINT
   					Numero_Texte														:= 2000+ L_Msg_Index;			// Class 2 Faultt
   			(*================================================================================================
   										Commutation Offset Uninitialized
   			==================================================================================================*)
   			ELSIF 	MIO_Axis.CommutationOffsetUninitializedFault THEN
   			 		L_Msg_Index													:= 350;							// Convert INT_To_DINT
   					Numero_Texte														:= 2000+ L_Msg_Index;			// Class 2 Faultt
   			(*================================================================================================
   										Invalid FPGA Image
   			==================================================================================================*)
   			ELSIF 	MIO_Axis.InvalidFPGAImageFault THEN
   			 		L_Msg_Index													:= 351;							// Convert INT_To_DINT
   					Numero_Texte														:= 2000+ L_Msg_Index;			// Class 2 Faultt
   			(*================================================================================================
   										Invalid Board Support Package
   			==================================================================================================*)
   			ELSIF 	MIO_Axis.InvalidBoardSupportPackageFault THEN
   			 		L_Msg_Index													:= 352;							// Convert INT_To_DINT
   					Numero_Texte														:= 2000+ L_Msg_Index;			// Class 2 Faultt
   			(*================================================================================================
   										Invalid Safety Firmware
   			==================================================================================================*)
   			ELSIF 	MIO_Axis.InvalidSafetyFirmwareFault THEN
   			 		L_Msg_Index													:= 353;							// Convert INT_To_DINT
   					Numero_Texte														:= 2000+ L_Msg_Index;			// Class 2 Faultt
   			(*================================================================================================
   										Power Board
   			==================================================================================================*)
   			ELSIF 	MIO_Axis.PowerBoardFault THEN
   			 		L_Msg_Index													:= 354;							// Convert INT_To_DINT
   					Numero_Texte														:= 2000+ L_Msg_Index;			// Class 2 Faultt
   			(*================================================================================================
   										Illegal Option Card
   			==================================================================================================*)
   			ELSIF 	MIO_Axis.IllegalOptionCardFault THEN
   			 		L_Msg_Index													:= 355;							// Convert INT_To_DINT
   					Numero_Texte														:= 2000+ L_Msg_Index;			// Class 2 Faultt
   			(*================================================================================================
   										Option Storage Checksum
   			==================================================================================================*)
   			ELSIF 	MIO_Axis.OptionStorageChecksumFault THEN
   			 		L_Msg_Index													:= 356;							// Convert INT_To_DINT
   					Numero_Texte														:= 2000+ L_Msg_Index;			// Class 2 Faultt
   			(*================================================================================================
   										Module Voltage Mismatch
   			==================================================================================================*)
   			ELSIF 	MIO_Axis.ModuleVoltageMismatchFault THEN
   			 		L_Msg_Index													:= 357;							// Convert INT_To_DINT
   					Numero_Texte														:= 2000+ L_Msg_Index;			// Class 2 Faultt
   			(*================================================================================================
   										Unknown Module
   			==================================================================================================*)
   			ELSIF 	MIO_Axis.UnknownModuleFault THEN
   			 		L_Msg_Index													:= 358;							// Convert INT_To_DINT
   					Numero_Texte														:= 2000+ L_Msg_Index;			// Class 2 Faultt
   			(*================================================================================================
   										Factory Configuration Error
   			==================================================================================================*)
   			ELSIF 	MIO_Axis.FactoryConfigurationErrorFault THEN
   			 		L_Msg_Index													:= 359;							// Convert INT_To_DINT
   					Numero_Texte														:= 2000+ L_Msg_Index;			// Class 2 Faultt
   			(*================================================================================================
   										Illegal Address
   			==================================================================================================*)
   			ELSIF 	MIO_Axis.IllegalAddressFault THEN
   			 		L_Msg_Index													:= 360;							// Convert INT_To_DINT
   					Numero_Texte														:= 2000+ L_Msg_Index;			// Class 2 Faultt
   			(*================================================================================================
   										Series Mismatch
   			==================================================================================================*)
   			ELSIF 	MIO_Axis.SeriesMismatchFault THEN
   			 		L_Msg_Index													:= 361;							// Convert INT_To_DINT
   					Numero_Texte														:= 2000+ L_Msg_Index;			// Class 2 Faultt
   			(*================================================================================================
   										Open Slot
   			==================================================================================================*)
   			ELSIF 	MIO_Axis.OpenSlotFault THEN
   			 		L_Msg_Index													:= 362;							// Convert INT_To_DINT
   					Numero_Texte														:= 2000+ L_Msg_Index;			// Class 2 Faultt
   			END_IF;
   
   	(*================================================================================================
   									APR Fault
   	==================================================================================================*)
   	ELSIF MIO_Axis.AxisFault.6 THEN
   
   			(*================================================================================================
   										APR FAULT
   			==================================================================================================*)
   					L_Msg_Index													:= 363;
   					Numero_Texte														:= 1000 + L_Msg_Index;		// Class 1 Fault
   	END_IF;
   
   	ER		:= TRUE;
   
   END_IF;
   
   IF MIO_Axis.AxisFault = 0 THEN
   	L_Msg_Index	:=0;
   	ER		:= FALSE;
   END_IF;
   (*================================================================================================
   										No Error Pending
   ==================================================================================================*)
   
END_ROUTINE
END_ADD_ON_INSTRUCTION
